// TIA Portal project "tasks 13.04" (V16)

(* hardware
DEVICE "S7-1200 station_1"  S7-1200 Station
   slot 0: "Rack_0"  S7-1200 Rack  Rack  V1.0
   slot 1: "PLC_1"  CPU 1217C DC/DC/DC  6ES7 217-1AG40-0XB0  V4.4
*)

// ===== PLC "PLC_1"  CPU 1217C DC/DC/DC =====

VAR_GLOBAL   // PLC tag table "Default tag table"
   "System_Byte" AT %MB1 : Byte;
   "FirstScan" AT %M1.0 : Bool;
   "DiagStatusUpdate" AT %M1.1 : Bool;
   "AlwaysTRUE" AT %M1.2 : Bool;
   "AlwaysFALSE" AT %M1.3 : Bool;
   "Clock_Byte" AT %MB0 : Byte;
   "Clock_10Hz" AT %M0.0 : Bool;
   "Clock_5Hz" AT %M0.1 : Bool;
   "Clock_2.5Hz" AT %M0.2 : Bool;
   "Clock_2Hz" AT %M0.3 : Bool;
   "Clock_1.25Hz" AT %M0.4 : Bool;
   "Clock_1Hz" AT %M0.5 : Bool;
   "Clock_0.625Hz" AT %M0.6 : Bool;
   "Clock_0.5Hz" AT %M0.7 : Bool;
   "Michal" AT %I0.0 : Bool;
   "Zosia" AT %Q0.0 : Bool;
   "x" AT %MD2 : Real;
   "y" AT %MD6 : Real;
   "z1" AT %MD10 : Real;
   "z2" AT %MD14 : Real;
   "z3" AT %MD18 : Real;
   "z4" AT %MD22 : Real;
   "WYNIK" AT %MD26 : Real;
   "Wynik2" AT %MD30 : Real;
   "licznik" AT %IW2 : UInt;
   "CzujnikSamochodow" AT %I0.1 : Bool;
   "byleco" AT %M36.0 : Bool;
   "Reset" AT %I0.2 : Bool;
   "t1" AT %M38.0 : LReal;
   "t2" AT %M46.0 : LReal;
   "t3" AT %M54.0 : LReal;
   "t4" AT %M62.0 : LReal;
   "wynikt" AT %M70.0 : LReal;
   "t5" AT %M78.0 : LReal;
   "t6" AT %M86.0 : LReal;
   "TemperatureF" AT %M94.0 : LReal;
   "TemperatureC" AT %M102.0 : LReal;
END_VAR

ORGANIZATION_BLOCK "Main"   // OB1, LAD, ProgramCycle
TITLE = "Main Program Sweep (Cycle)"
{ S7_Optimized_Access := 'TRUE' }
VERSION : 0.1
   VAR_INPUT
      Initial_Call : Bool;   // Initial call of this OB
      Remanence : Bool;   // =True, if remanent data are available
   END_VAR
   VAR_TEMP   // added for the SCL form of the ladder/FBD networks
      _w1 : Bool;
   END_VAR
BEGIN

REGION Network 1
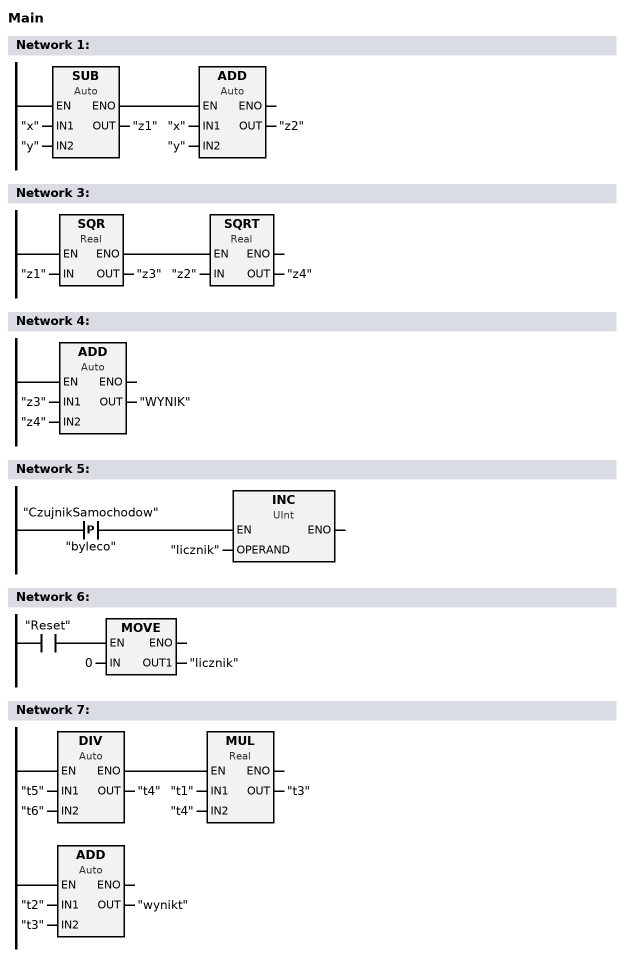
   RUNG wire#powerrail
      Sub(in1 := "x", in2 := "y", out => "z1")
      Add(in1 := "x", in2 := "y", out => "z2")
   END_RUNG
   // the same network as SCL:
   "z1" := "x" - "y";
   "z2" := "x" + "y";
END_REGION

REGION Network 2 (SCL)
   "Wynik2" := ("x" - "y") * ("x" - "y") + SQRT("x" + "y");
END_REGION

REGION Network 3
   "z3" := SQR("z1");
   "z4" := SQRT("z2");
END_REGION

REGION Network 4
   RUNG wire#powerrail
      Add(in1 := "z3", in2 := "z4", out => "WYNIK")
   END_RUNG
   // the same network as SCL:
   "WYNIK" := "z3" + "z4";
END_REGION

REGION Network 5
   RUNG wire#powerrail
      P_Contact(operand := "CzujnikSamochodow", bit := "byleco")
      { S7_Templates := "DestType := UInt" } Inc( "licznik" )
   END_RUNG
   // the same network as SCL:
   #_w1 := "CzujnikSamochodow" AND NOT "byleco";   // rising edge of "CzujnikSamochodow"
   "byleco" := "CzujnikSamochodow";
   IF #_w1 THEN "licznik" := "licznik" + 1; END_IF;
END_REGION

REGION Network 6
   RUNG wire#powerrail
      Contact( "Reset" )
      Move(in := 0, out1 => "licznik")
   END_RUNG
   // the same network as SCL:
   IF "Reset" THEN "licznik" := 0; END_IF;
END_REGION

REGION Network 7
   RUNG wire#powerrail
      Div(in1 := "t5", in2 := "t6", out => "t4")
      { S7_Templates := "SrcType := Real" } Mul(in1 := "t1", in2 := "t4", out => "t3")
   END_RUNG
   RUNG wire#powerrail
      Add(in1 := "t2", in2 := "t3", out => "wynikt")
   END_RUNG
   // the same network as SCL:
   "t4" := "t5" / "t6";
   "t3" := "t1" * "t4";
   "wynikt" := "t2" + "t3";
END_REGION

REGION Network 8 (SCL)
   "TemperatureF" := 32.0 + 1.8 * "TemperatureC";
END_REGION
END_ORGANIZATION_BLOCK